Fanuc KAREL source: kb00191.KL

-- PROVISIONAL review KL for V1013-1; original PC SHA256 4fb4efa25f4995fcfc4c9064f9b83ec41c6f72af3e1d5be29d2ee45a34584f08
-- Incomplete behavior may be omitted. Consult companion uncertainty JSON. Do not deploy.
PROGRAM KB00191
%NOLOCKGROUP
BEGIN
  -- UNRESOLVED_PC offsets 5-14; opcodes 3F,75
  -- UNRESOLVED_PC offsets 19-26; opcodes 9D,23
  -- UNRESOLVED_PC offsets 31-38; opcodes 9D,23
  -- UNRESOLVED_PC offsets 43-67; opcodes 27,22,2A,22,22,31
  -- UNRESOLVED_PC offsets 72-76; opcodes 7F
END KB00191
